FUNCTION HMI_Component : INT

VAR_INPUT
	Act_Pnl: INT; //The Active HMI Screen Reference Number
	Loc_Pnl: INT; //THe HMI Screen that the Component is located, 0=Universal component (located on all screens)
END_VAR

VAR

END_VAR

VAR_IN_OUT
	COMP:TS_Component;
END_VAR

//Section that controls pushbutton state logic
	IF ( (Loc_Pnl=0 OR ACT_Pnl=Loc_Pnl) AND COMP.invisible=0 AND COMP.display_state>0  AND COMP.B_TYPE<10 ) THEN
		IF (COMP.B_TYPE = 0) THEN (*Momentary button type*) 
			IF (COMP.Active = 0) THEN
				COMP.State:=0;
				COMP.run_status:=0;
			ELSIF (COMP.Active = 1 AND COMP.run_status = 0) THEN
				COMP.State:=1;
				COMP.run_status:=1;
			ELSIF (COMP.Active = 1 AND COMP.run_status = 1) THEN
				COMP.State:=0;
				COMP.Active:=0;
			END_IF
		ELSIF (COMP.B_TYPE = 1) THEN (*Maintained button type*)
			IF (COMP.Active = 0) THEN
				COMP.State:=0;
				COMP.run_status:=0;
			ELSIF (COMP.Active = 1) THEN
				COMP.State:=1;
				COMP.run_status:=1;
			END_IF
		ELSIF (COMP.B_TYPE = 2) THEN (*Toggle button type*)
			IF (COMP.Active = 0) THEN
				COMP.run_status:=0;
			ELSIF (COMP.Active = 1 AND COMP.run_status = 0) THEN
				IF (COMP.State=0) THEN
					COMP.State:=1;
				ELSE
					COMP.State:=0;
				END_IF
				COMP.run_status:=1;
			ELSE
				COMP.Active:=0;
			END_IF
		ELSE
			COMP.State:=0;
			COMP.Active:=FALSE;
		END_IF
	ELSE
		COMP.State:=FALSE;
		COMP.Active:=FALSE;
	END_IF
	
//Section that controls the displayed image for the HMI Component
	IF ((Loc_Pnl=0 OR ACT_Pnl=Loc_Pnl) AND COMP.invisible=0) THEN
		IF (COMP.size=0) THEN
			IF (COMP.display_state=0) THEN
				COMP.bitmap_ID:='ImagePool.PB_GY_125_100';
			ELSIF (COMP.display_state=1) THEN
				COMP.bitmap_ID:='ImagePool.PB_BU_125_100';
			ELSIF (COMP.display_state=2) THEN
				COMP.bitmap_ID:='ImagePool.PB_GN_125_100';
			ELSIF (COMP.display_state=3) THEN
				COMP.bitmap_ID:='ImagePool.PB_RD_125_100';
			ELSE
				COMP.bitmap_ID:='ImagePool.PB_GY_125_100';
			END_IF
		ELSIF (COMP.size=1) THEN
			IF (COMP.display_state=0) THEN
				COMP.bitmap_ID:='ImagePool.PB_GY_75_75';
			ELSIF (COMP.display_state=1) THEN
				COMP.bitmap_ID:='ImagePool.PB_BU_75_75';
			ELSIF (COMP.display_state=2) THEN
				COMP.bitmap_ID:='ImagePool.PB_GN_75_75';
			ELSIF (COMP.display_state=3) THEN
				COMP.bitmap_ID:='ImagePool.PB_RD_75_75';
			ELSE
				COMP.bitmap_ID:='ImagePool.PB_GY_75_75';
			END_IF
		ELSIF (COMP.size=2) THEN
			IF (COMP.display_state=0) THEN
				COMP.bitmap_ID:='ImagePool.PB_GY_160_75';
			ELSIF (COMP.display_state=1) THEN
				COMP.bitmap_ID:='ImagePool.PB_BU_160_75';
			ELSIF (COMP.display_state=2) THEN
				COMP.bitmap_ID:='ImagePool.PB_GN_160_75';
			ELSIF (COMP.display_state=3) THEN
				COMP.bitmap_ID:='ImagePool.PB_RD_160_75';
			ELSE
				COMP.bitmap_ID:='ImagePool.PB_GY_160_75';
			END_IF
		ELSIF (COMP.size=3) THEN
			IF (COMP.display_state=0) THEN
				COMP.bitmap_ID:='ImagePool.PB_GY_250_75';
			ELSIF (COMP.display_state=1) THEN
				COMP.bitmap_ID:='ImagePool.PB_BU_250_75';
			ELSIF (COMP.display_state=2) THEN
				COMP.bitmap_ID:='ImagePool.PB_GN_250_75';
			ELSIF (COMP.display_state=3) THEN
				COMP.bitmap_ID:='ImagePool.PB_RD_250_75';
			ELSE
				COMP.bitmap_ID:='ImagePool.PB_GY_250_75';
			END_IF
		ELSIF (COMP.size=10) THEN
			IF (COMP.display_state=0) THEN
				COMP.bitmap_ID:='ImagePool.IN_BU_300_50';
			ELSIF (COMP.display_state=1) THEN
				COMP.bitmap_ID:='ImagePool.IN_GN_300_50';
			ELSIF (COMP.display_state=2) THEN
				COMP.bitmap_ID:='ImagePool.IN_RD_300_50';
			ELSIF (COMP.display_state=3) THEN
				COMP.bitmap_ID:='ImagePool.IN_YL_300_50';
			ELSIF (COMP.display_state=4) THEN
				COMP.bitmap_ID:='ImagePool.IN_GY_300_50';
			ELSIF (COMP.display_state=5) THEN
				COMP.bitmap_ID:='ImagePool.IN_RR_300_50';
			ELSIF (COMP.display_state=6) THEN
				COMP.bitmap_ID:='ImagePool.IN_RY_300_50';
			ELSIF (COMP.display_state=7) THEN
				COMP.bitmap_ID:='ImagePool.IN_YR_300_50';
			ELSIF (COMP.display_state=8) THEN
				COMP.bitmap_ID:='ImagePool.IN_CL_61_40';
			ELSE 
				COMP.bitmap_ID:='ImagePool.IN_RR_300_50';
			END_IF
		ELSIF (COMP.size=11) THEN
			IF (COMP.display_state=0) THEN
				COMP.bitmap_ID:='ImagePool.IN_BU_61_40';
			ELSIF (COMP.display_state=1) THEN
				COMP.bitmap_ID:='ImagePool.IN_GN_61_40';
			ELSIF (COMP.display_state=2) THEN
				COMP.bitmap_ID:='ImagePool.IN_RD_61_40';
			ELSIF (COMP.display_state=3) THEN
				COMP.bitmap_ID:='ImagePool.IN_YL_61_40';
			ELSIF (COMP.display_state=4) THEN
				COMP.bitmap_ID:='ImagePool.IN_GY_61_40';
			ELSIF (COMP.display_state=5) THEN
				COMP.bitmap_ID:='ImagePool.IN_RR_61_40';
			ELSIF (COMP.display_state=6) THEN
				COMP.bitmap_ID:='ImagePool.IN_RY_61_40';
			ELSIF (COMP.display_state=7) THEN
				COMP.bitmap_ID:='ImagePool.IN_YR_61_40';
			ELSIF (COMP.display_state=8) THEN
				COMP.bitmap_ID:='ImagePool.IN_CL_61_40';
			ELSE 
				COMP.bitmap_ID:='ImagePool.IN_RR_61_40';
			END_IF
		END_IF
	END_IF

END_FUNCTION

(* stored: Version 1.1.0.1, ProductVersion 3.1.4020.12
   POU HMI_Component: Id {d84bd541-94ef-4c60-b9b4-6ff9186af438}, SpecialFunc None *)
